{attribute 'GeneratedUsingTerminal: EL1262-0000-0002'}
{attribute addProperty BoxType "EL1262-0000-0002"}
{attribute addProperty Id "Ch2_InputAT %I*BOOL1"}
{attribute addProperty CRC "2024646924"}
{attribute addProperty Size "1"}
TYPE Ch2_Input_78ADA90C EXTENDS InputBase_8311D824 :
STRUCT
	{attribute addProperty Name "Ch2_Input"}
	Ch2_Input AT %I* : BOOL;
END_STRUCT
END_TYPE

(* stored: Version 1.2.0.0, ProductVersion 3.1.4024.9
   DUT Ch2_Input_78ADA90C: Id {58c3fd23-3396-4eea-828b-732e12d52270} *)
